TYPE ST_FunctionData :
(**************************************************************************************
 * 	Application		:	BoxControl Framework
 *	Revision		:	$Revision: 404529 $
 *	Revision date	:	$Date: 2018-04-23 08:21:38 +0200 (Mo., 23 Apr 2018) $
 *	Last changed by	:	$Author: b7bolm $
 *	URL				:	$URL: http://almscdc.swisslog.com/repo/SWPD/Development/BoxControlFramework/20_Release/trunk/01_Software/BCF/BCF/JumpStart/20_Product/10_App/12_E_Functions/10_Lib/10_Conv/01_DUTs/ST_FunctionData.TcDUT $
 *
 *	Purpose			:	Function data
 *
 * ------------------------------------------------------------------------------------
 *	Copyright Swisslog [IP AG], Switzerland. All rights reserved.
 * 
 * ------------------------------------------------------------------------------------
 *	
 * 	Revision History: 
 *
 * 	VERSION			DATE			INITIALS			DESCRIPTION
 *	0.1				01.01.2001		swl					Example
 *
 **************************************************************************************)
STRUCT
	Init				: BOOL; // Initialized
	InitRunning			: BOOL; // Init ongoing
	OperationState		: ST_PositionState; // Information about the state
	AddOn				: ST_AddOnResult; // Result form external addons
	MemberList			: ST_FunctionMemberList; // List of members belonging to this function
	ErrorData			: ST_FunctionErrorStruct; // Error structure
	AddOnData			: ST_AddOnData; // Specific addon data structs
	ControlRequest		: ST_ControlRequest; // Control request
END_STRUCT
END_TYPE

(* stored: Version 1.1.0.1, ProductVersion 3.1.4022.12
   DUT ST_FunctionData: Id {471cc2d4-3435-4bb4-8bf6-10ea2dc799ac} *)
